(* CoDeSys 2.3 export: PUMP.EXP *)

(* POU PRG/Pump, CFC *)
PROGRAM Pump
VAR
END_VAR
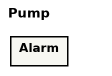
_CFC_ (* Continuous Function Chart, elements in execution order *)
#0 Alarm()
_END_CFC_
(* the same logic as Structured Text *)
Alarm();
END_PROGRAM
